PROGRAM prgSystem
VAR_IN_OUT
	iTaskIdx		: DINT;
	bFirstCycle		: BOOL;
END_VAR

// Scan Control
bFirstCycle := TwinCAT_SystemInfoVarList._TaskInfo[iTaskIdx].FirstCycle;

// Mode Control
gvlMotion.autoMode := NOT gvlMotion.manualMode;

END_PROGRAM

(* stored: Version 1.1.0.1, ProductVersion 3.1.4024.12
   POU prgSystem: Id {4bcb5386-353b-4a56-9a7b-592b4f1aab8a}, SpecialFunc None *)
